// Block: A0303_Sostegno_PERS

DATA_BLOCK A0303_Sostegno_PERS
VERSION : 0.1
   NON_RETAIN
   VAR
      Par : Struct
         Testa : Struct
            Ax : Positioning_DOL_Machine_Par;
            Ax_Pers : Positioning_DOL_Machine_Pers_Data;
            Enc : PosFbk_RTN;
         END_STRUCT;
         Coda : Struct
            Ax : Positioning_DOL_Machine_Par;
            Ax_Pers : Positioning_DOL_Machine_Pers_Data;
            Enc : PosFbk_RTN;
         END_STRUCT;
      END_STRUCT;
      Par_Mach : Struct
         RestPosition : LReal;
         ToleranceWindow : LReal;
         PosTimeout : Time;
      END_STRUCT;
   END_VAR

BEGIN
   // No initialization required
END_DATA_BLOCK
